{attribute 'GeneratedUsingTerminal: ER2008-0001-0018'}
{attribute addProperty BoxType "ER2008-0001-0018"}
{attribute addProperty Id "WcStateAT %I*BOOL1"}
{attribute addProperty CRC "187373305"}
{attribute addProperty Size "1"}
TYPE WcState_0B2B16F9 :
STRUCT
	{attribute addProperty Name "WcState"}
	WcState AT %I* : BOOL;
END_STRUCT
END_TYPE

(* stored: Version 1.2.0.0, ProductVersion 3.1.4024.9
   DUT WcState_0B2B16F9: Id {c9d2f0be-add4-4326-9a96-2f7e58d33265} *)
